FUNCTION_BLOCK FB_SaMElementAborting EXTENDS FB_SaMElement
VAR
END_VAR

END_FUNCTION_BLOCK

(* stored: Version 1.1.0.1
   POU FB_SaMElementAborting: Id {c7d1042c-68f1-06d1-0ebb-5647496def75}, SpecialFunc None *)
